{attribute 'linkalways'} 
{attribute 'no_explicit_call' := 'This FB is a CLASS and must be accessed using methods or properties'}
{attribute 'enable_dynamic_creation'}
FUNCTION_BLOCK _ETcVnMatchTemplateWalshOptions EXTENDS EnumDatatypeBase
VAR
	localData : ETcVnMatchTemplateWalshOptions;
	activeData : REFERENCE TO ETcVnMatchTemplateWalshOptions;
	enumBaseDatatype : _UDINT(localData);
END_VAR

METHOD PRIVATE AddLocalEnumeration
VAR_INPUT
	Enumeration : T_MAXSTRING;
	Value : ETcVnMatchTemplateWalshOptions;
END_VAR
AddEnumeration(Enumeration, Value);
END_METHOD

PROPERTY PUBLIC Address : PVOID
GET
Address := ADR(activeData);
END_GET
END_PROPERTY

METHOD PUBLIC ClearReference
VAR_INPUT
END_VAR
activeData REF= localData;
SetBaseDatatypeReference();
END_METHOD

METHOD PUBLIC Clone : I_Datatype
VAR
    pClone : POINTER TO _ETcVnMatchTemplateWalshOptions;
END_VAR
pClone := __NEW(_ETcVnMatchTemplateWalshOptions(InitialValue := Value));
Clone := pClone^;
END_METHOD

METHOD FB_init : BOOL
VAR_INPUT
	bInitRetains : BOOL; // if TRUE, the retain variables are initialized (warm start / cold start)
	bInCopyCode : BOOL;  // if TRUE, the instance afterwards gets moved into the copy code (online change)
	InitialValue : ETcVnMatchTemplateWalshOptions;
END_VAR
localData := InitialValue;
AddBaseDatatype(enumBaseDatatype);
ClearReference();

AddLocalEnumeration('TCVN_MTWO_NONE', ETcVnMatchTemplateWalshOptions.TCVN_MTWO_NONE);
AddLocalEnumeration('TCVN_MTWO_NORMED', ETcVnMatchTemplateWalshOptions.TCVN_MTWO_NORMED);
AddLocalEnumeration('TCVN_MTWO_SKIP_DC', ETcVnMatchTemplateWalshOptions.TCVN_MTWO_SKIP_DC);
END_METHOD

PROPERTY PUBLIC Identifier : T_MAXSTRING
GET
Identifier := 'ETcVnMatchTemplateWalshOptions';
END_GET
END_PROPERTY

METHOD IsEnumeratorValueEqual : BOOL
VAR_INPUT
	Enumerator : I_KeyValueForwardEnumerator;
END_VAR
VAR
	storedValue : ETcVnMatchTemplateWalshOptions;
END_VAR
IF NOT Enumerator.TryGet(storedValue) THEN
	RETURN;
END_IF

IsEnumeratorValueEqual := storedValue = activeData;
END_METHOD

METHOD PUBLIC MakeReferenceTo
VAR_INPUT
	ReferenceTarget : REFERENCE TO ETcVnMatchTemplateWalshOptions;
END_VAR
activeData REF= ReferenceTarget;
SetBaseDatatypeReference();
END_METHOD

METHOD PROTECTED SetBaseDatatypeReference
VAR_INPUT
END_VAR
enumBaseDatatype.MakeReferenceTo(activeData);
END_METHOD

PROPERTY PUBLIC Size : UDINT
GET
Size := SIZEOF(activeData);
END_GET
END_PROPERTY

METHOD TryMakeReferenceTo : BOOL
VAR_INPUT
	Target : I_Datatype;
END_VAR
VAR
	pTargetData : POINTER TO ETcVnMatchTemplateWalshOptions;
END_VAR
IF NOT IsEquivalentTo(Target) THEN
	RETURN;
END_IF

pTargetData := Target.Address;
activeData REF= pTargetData^;
SetBaseDatatypeReference();
TryMakeReferenceTo := TRUE;
END_METHOD

PROPERTY PUBLIC Value : ETcVnMatchTemplateWalshOptions
GET
Value := activeData;
END_GET
SET
activeData := Value;
END_SET
END_PROPERTY

END_FUNCTION_BLOCK

(* stored: Version 1.1.0.1, ProductVersion 3.1.4026.13
   POU _ETcVnMatchTemplateWalshOptions: Id {b604166e-e1af-0f50-167f-55cc951c4741}, SpecialFunc None
   Folder Core: Id {896fd416-fb40-0e0d-09fc-bc8d658ba512}
   Folder Protected: Id {80ec0409-9b19-062b-35a0-2be4e8429ec2}
   Folder Customize: Id {ff83f639-6a90-0131-15fb-81f8b58e38ac}
   Folder Constructor: Id {f7dbc0fc-3dc5-0780-395b-9146fe6fcbb4}
   Folder Private: Id {7982ffdd-2d54-0876-2b0f-d14dfcaed7d2}
   Folder Protected: Id {741802c4-ffa0-0432-2a95-3662d254a2db}
   Method AddLocalEnumeration: Id {142fcdc2-f83b-03fd-07c7-e01a5b07b306}
   Property Address: Id {3eb413e1-d4a9-0e97-08b6-af5886181cbb}
   Get Get: Id {940b6f6d-3c26-0677-337c-bdf71309718f}
   Method ClearReference: Id {f4afca31-8476-07e6-3f3f-8f1452997ecc}
   Method Clone: Id {112676a4-1db2-086c-330a-da3466cad923}
   Method FB_init: Id {6a8ab18c-76d3-0221-3729-cdbc7487a1f7}
   Property Identifier: Id {917208f0-e387-0890-059f-f3509d4afb86}
   Get Get: Id {e97856d7-db28-0dd4-1cde-bc4a86dce6f7}
   Method IsEnumeratorValueEqual: Id {ecf6061f-2833-04d6-04b4-69cea1e614e5}
   Method MakeReferenceTo: Id {bf621564-85a4-0703-0036-d5f5568f1e8b}
   Method SetBaseDatatypeReference: Id {1c6e0cec-f739-0ddf-06b7-0447c27642c5}
   Property Size: Id {788ccac2-a2bc-0aac-2380-77a8e6b7b599}
   Get Get: Id {83c092a4-4188-0b74-1f83-3949a1008c9f}
   Method TryMakeReferenceTo: Id {927e0eb6-135f-0b6b-207f-5ec46fff9de2}
   Property Value: Id {54b145ee-5f2d-0e01-1368-dd888ea14f79}
   Get Get: Id {96619721-ddaa-049b-0513-c5b8a0cb60d2}
   Set Set: Id {3e167177-3c7e-0bf7-17c3-dc0288c59f0d} *)
